{region '#Template'}
	{attribute 'Version' := '1.0.0.0'}
	{attribute 'Tags' := '"LCID": "1031", "Text": "H, General, HtgCir, Operating mode"'}
	{attribute 'Tags' := '"LCID": "1033", "Text": "H, General, HtgCir, Operating mode"'}
	{attribute 'Description' := '"LCID": "1031", "Text": "Betriebsart"'}
	{attribute 'Description' := '"LCID": "1033", "Text": "Operating mode"'}
{endregion}
FUNCTION_BLOCK FB_BA_H_OpMod EXTENDS FB_BA_View
VAR_INPUT
	bDst					: BOOL;
	bHtgLmt					: BOOL;
	bTWthLowLimit			: BOOL;
END_VAR
VAR_OUTPUT
	eOpMod					: E_BA_EnergyLvl;
	bRls					: BOOL;
END_VAR
VAR_INPUT CONSTANT
	OpModMan				: FB_BA_MV_Op;
	Sched					: FB_BA_SchedM;
	OpModPr					: FB_BA_MV_Op;								 
	Rls						: FB_BA_BV_Op;
END_VAR
VAR
	OpModSwi				: FB_BA_PrioSwi_UDI08;
	RlsMMux					: FB_BA_MMUX_B04;
END_VAR

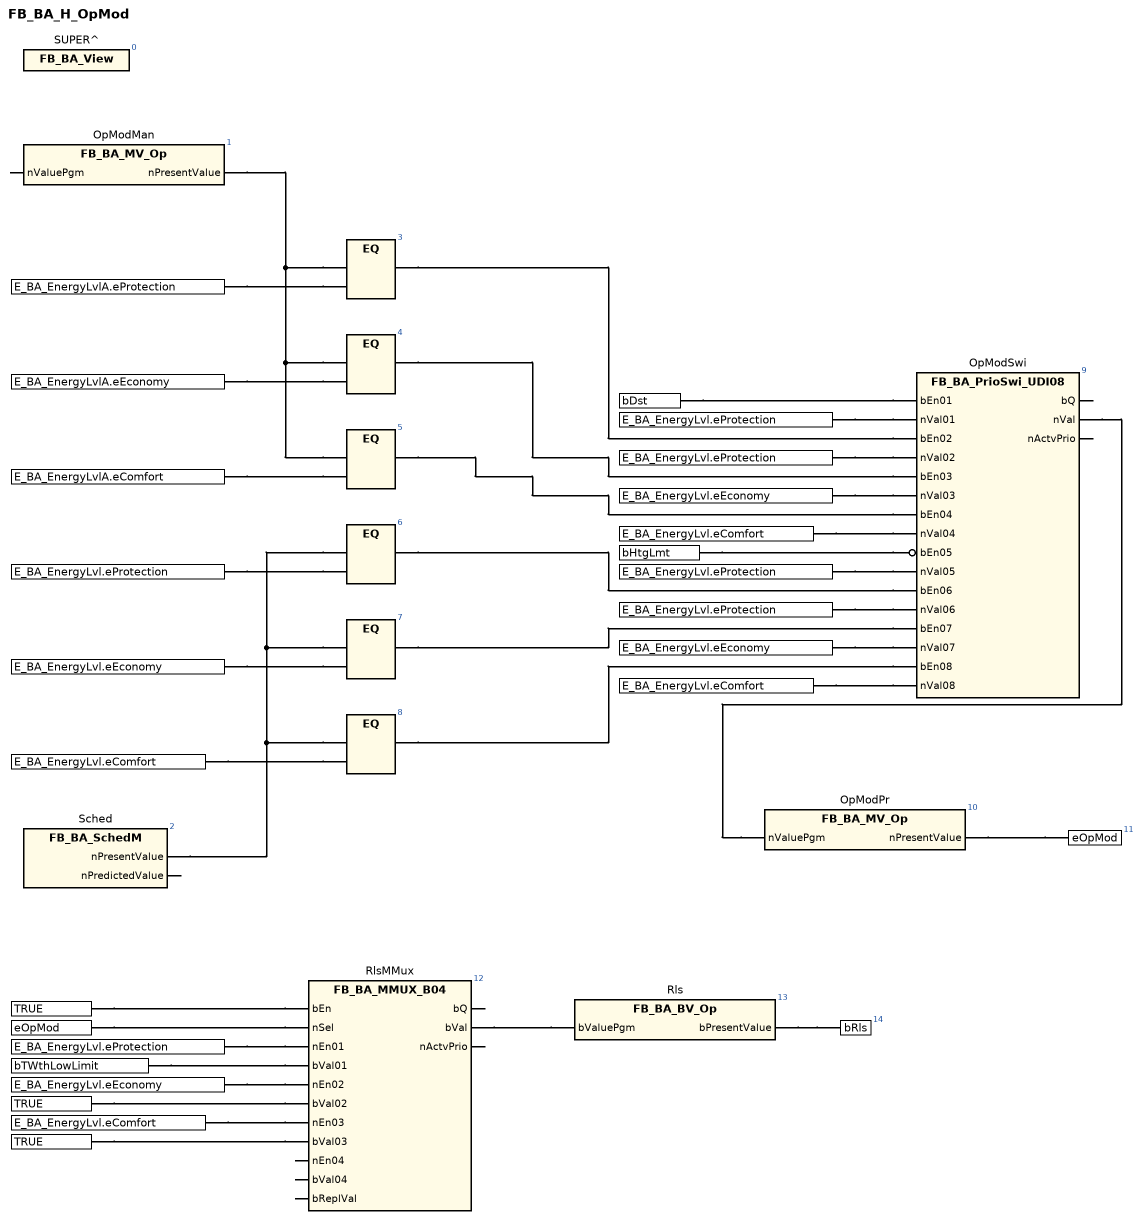
SUPER^(); // FB_BA_View
OpModMan(); // FB_BA_MV_Op
Sched(); // FB_BA_SchedM
OpModSwi(
    bEn01 := bDst,
    nVal01 := E_BA_EnergyLvl.eProtection,
    bEn02 := OpModMan.nPresentValue = E_BA_EnergyLvlA.eProtection,
    nVal02 := E_BA_EnergyLvl.eProtection,
    bEn03 := OpModMan.nPresentValue = E_BA_EnergyLvlA.eEconomy,
    nVal03 := E_BA_EnergyLvl.eEconomy,
    bEn04 := OpModMan.nPresentValue = E_BA_EnergyLvlA.eComfort,
    nVal04 := E_BA_EnergyLvl.eComfort,
    bEn05 := NOT bHtgLmt,
    nVal05 := E_BA_EnergyLvl.eProtection,
    bEn06 := Sched.nPresentValue = E_BA_EnergyLvl.eProtection,
    nVal06 := E_BA_EnergyLvl.eProtection,
    bEn07 := Sched.nPresentValue = E_BA_EnergyLvl.eEconomy,
    nVal07 := E_BA_EnergyLvl.eEconomy,
    bEn08 := Sched.nPresentValue = E_BA_EnergyLvl.eComfort,
    nVal08 := E_BA_EnergyLvl.eComfort); // FB_BA_PrioSwi_UDI08
OpModPr(nValuePgm := OpModSwi.nVal); // FB_BA_MV_Op
eOpMod := OpModPr.nPresentValue;
RlsMMux(
    bEn := TRUE,
    nSel := eOpMod,
    nEn01 := E_BA_EnergyLvl.eProtection,
    bVal01 := bTWthLowLimit,
    nEn02 := E_BA_EnergyLvl.eEconomy,
    bVal02 := TRUE,
    nEn03 := E_BA_EnergyLvl.eComfort,
    bVal03 := TRUE); // FB_BA_MMUX_B04
Rls(bValuePgm := RlsMMux.bVal); // FB_BA_BV_Op
bRls := Rls.bPresentValue;

METHOD FB_init : BOOL
VAR_INPUT
	bInitRetains : BOOL; // if TRUE, the retain variables are initialized (warm start / cold start)
	bInCopyCode : BOOL;  // if TRUE, the instance afterwards gets moved into the copy code (online change)
END_VAR
OpModMan.iParent		:= THIS^;
OpModMan.iLabel			:= LblCmpHeating.H_OpMod_OpModMan;							
OpModMan.sObjectName	:= '{Idx=01}';								 	 
OpModMan.aStateText[1]	:= txtEvent_Auto;
OpModMan.aStateText[2]	:= txtEvent_Protection;
OpModMan.aStateText[3]	:= txtEvent_Economy;
OpModMan.aStateText[4]	:= txtEvent_Comfort;
OpModMan.nValueRm		:= 1;

OpModPr.iParent			:= THIS^;
OpModPr.iLabel			:= LblCmpHeating.H_OpMod_OpModPr;							
OpModPr.sObjectName		:= '{Idx=01}';								 	 
OpModPr.aStateText[1]	:= txtEvent_Protection; 
OpModPr.aStateText[2]	:= txtEvent_Economy; 
OpModPr.aStateText[3]	:= txtEvent_Comfort; 
OpModPr.nValueRm		:= 1;

Rls.iParent				:= THIS^;
Rls.iLabel				:= LblCmpHeating.H_OpMod_Rls;	
Rls.sObjectName			:= '{Idx=01}';								 	 
Rls.sInactiveText		:= txtEvent_Off;
Rls.sActiveText			:= txtEvent_On;	
Rls.bValueRm			:= FALSE;								
Rls.eToggleMode 		:= E_BA_ToggleMode.eSwitch;	

Sched.iParent											:= THIS^;
Sched.iLabel											:= LblCmpHeating.H_OpMod_Sched;							
Sched.sObjectName										:= '{Idx=01}';								 	 
Sched.aStateText[1]										:= txtEvent_Protection;
Sched.aStateText[2]										:= txtEvent_Economy;
Sched.aStateText[3]										:= txtEvent_Comfort;
Sched.nPredictTime										:= 0;
Sched.nDefaultValue										:= E_BA_EnergyLvl.eProtection;
Sched.bWriteWeekly										:= FALSE;
//	Monday
Sched.aWeek[E_BA_Weekday.eMonday,1].eState				:= E_BA_SchedEntryState.eValue;
Sched.aWeek[E_BA_Weekday.eMonday,1].uValue.udiVal		:= E_BA_EnergyLvl.eComfort;
Sched.aWeek[E_BA_Weekday.eMonday,1].stTime.nHour		:= 6;
Sched.aWeek[E_BA_Weekday.eMonday,1].stTime.nMinute		:= 0;
Sched.aWeek[E_BA_Weekday.eMonday,1].stTime.nSecond		:= 0;
Sched.aWeek[E_BA_Weekday.eMonday,2].eState				:= E_BA_SchedEntryState.eValue;
Sched.aWeek[E_BA_Weekday.eMonday,2].uValue.udiVal		:= E_BA_EnergyLvl.eEconomy;
Sched.aWeek[E_BA_Weekday.eMonday,2].stTime.nHour		:= 20;
Sched.aWeek[E_BA_Weekday.eMonday,2].stTime.nMinute		:= 0;
Sched.aWeek[E_BA_Weekday.eMonday,2].stTime.nSecond		:= 0;
Sched.aWeek[E_BA_Weekday.eMonday,3].eState				:= E_BA_SchedEntryState.eValue;
Sched.aWeek[E_BA_Weekday.eMonday,3].uValue.udiVal		:= E_BA_EnergyLvl.eProtection;
Sched.aWeek[E_BA_Weekday.eMonday,3].stTime.nHour		:= 0;
Sched.aWeek[E_BA_Weekday.eMonday,3].stTime.nMinute		:= 0;
Sched.aWeek[E_BA_Weekday.eMonday,3].stTime.nSecond		:= 0;
//	Tuesday
Sched.aWeek[E_BA_Weekday.eTuesday,1].eState				:= E_BA_SchedEntryState.eValue;
Sched.aWeek[E_BA_Weekday.eTuesday,1].uValue.udiVal		:= E_BA_EnergyLvl.eComfort;
Sched.aWeek[E_BA_Weekday.eTuesday,1].stTime.nHour		:= 6;
Sched.aWeek[E_BA_Weekday.eTuesday,1].stTime.nMinute		:= 0;
Sched.aWeek[E_BA_Weekday.eTuesday,1].stTime.nSecond		:= 0;
Sched.aWeek[E_BA_Weekday.eTuesday,2].eState				:= E_BA_SchedEntryState.eValue;
Sched.aWeek[E_BA_Weekday.eTuesday,2].uValue.udiVal		:= E_BA_EnergyLvl.eEconomy;
Sched.aWeek[E_BA_Weekday.eTuesday,2].stTime.nHour		:= 20;
Sched.aWeek[E_BA_Weekday.eTuesday,2].stTime.nMinute		:= 0;
Sched.aWeek[E_BA_Weekday.eTuesday,2].stTime.nSecond		:= 0;
Sched.aWeek[E_BA_Weekday.eTuesday,3].eState				:= E_BA_SchedEntryState.eValue;
Sched.aWeek[E_BA_Weekday.eTuesday,3].uValue.udiVal		:= E_BA_EnergyLvl.eProtection;
Sched.aWeek[E_BA_Weekday.eTuesday,3].stTime.nHour		:= 0;
Sched.aWeek[E_BA_Weekday.eTuesday,3].stTime.nMinute		:= 0;
Sched.aWeek[E_BA_Weekday.eTuesday,3].stTime.nSecond		:= 0;
//	Wednesday
Sched.aWeek[E_BA_Weekday.eWednesday,1].eState			:= E_BA_SchedEntryState.eValue;
Sched.aWeek[E_BA_Weekday.eWednesday,1].uValue.udiVal	:= E_BA_EnergyLvl.eComfort;
Sched.aWeek[E_BA_Weekday.eWednesday,1].stTime.nHour		:= 6;
Sched.aWeek[E_BA_Weekday.eWednesday,1].stTime.nMinute	:= 0;
Sched.aWeek[E_BA_Weekday.eWednesday,1].stTime.nSecond	:= 0;
Sched.aWeek[E_BA_Weekday.eWednesday,2].eState			:= E_BA_SchedEntryState.eValue;
Sched.aWeek[E_BA_Weekday.eWednesday,2].uValue.udiVal	:= E_BA_EnergyLvl.eEconomy;
Sched.aWeek[E_BA_Weekday.eWednesday,2].stTime.nHour		:= 20;
Sched.aWeek[E_BA_Weekday.eWednesday,2].stTime.nMinute	:= 0;
Sched.aWeek[E_BA_Weekday.eWednesday,2].stTime.nSecond	:= 0;
Sched.aWeek[E_BA_Weekday.eWednesday,3].eState			:= E_BA_SchedEntryState.eValue;
Sched.aWeek[E_BA_Weekday.eWednesday,3].uValue.udiVal	:= E_BA_EnergyLvl.eProtection;
Sched.aWeek[E_BA_Weekday.eWednesday,3].stTime.nHour		:= 0;
Sched.aWeek[E_BA_Weekday.eWednesday,3].stTime.nMinute	:= 0;
Sched.aWeek[E_BA_Weekday.eWednesday,3].stTime.nSecond	:= 0;
//	Thursday
Sched.aWeek[E_BA_Weekday.eThursday,1].eState			:= E_BA_SchedEntryState.eValue;
Sched.aWeek[E_BA_Weekday.eThursday,1].uValue.udiVal		:=E_BA_EnergyLvl.eComfort;
Sched.aWeek[E_BA_Weekday.eThursday,1].stTime.nHour		:= 6;
Sched.aWeek[E_BA_Weekday.eThursday,1].stTime.nMinute	:= 0;
Sched.aWeek[E_BA_Weekday.eThursday,1].stTime.nSecond	:= 0;
Sched.aWeek[E_BA_Weekday.eThursday,2].eState			:= E_BA_SchedEntryState.eValue;
Sched.aWeek[E_BA_Weekday.eThursday,2].uValue.udiVal		:= E_BA_EnergyLvl.eEconomy;
Sched.aWeek[E_BA_Weekday.eThursday,2].stTime.nHour		:= 20;
Sched.aWeek[E_BA_Weekday.eThursday,2].stTime.nMinute	:= 0;
Sched.aWeek[E_BA_Weekday.eThursday,2].stTime.nSecond	:= 0;
Sched.aWeek[E_BA_Weekday.eThursday,3].eState			:= E_BA_SchedEntryState.eValue;
Sched.aWeek[E_BA_Weekday.eThursday,3].uValue.udiVal		:= E_BA_EnergyLvl.eProtection;
Sched.aWeek[E_BA_Weekday.eThursday,3].stTime.nHour		:= 0;
Sched.aWeek[E_BA_Weekday.eThursday,3].stTime.nMinute	:= 0;
Sched.aWeek[E_BA_Weekday.eThursday,3].stTime.nSecond	:= 0;
//	Friday
Sched.aWeek[E_BA_Weekday.eFriday,1].eState				:= E_BA_SchedEntryState.eValue;
Sched.aWeek[E_BA_Weekday.eFriday,1].uValue.udiVal		:= E_BA_EnergyLvl.eComfort;
Sched.aWeek[E_BA_Weekday.eFriday,1].stTime.nHour		:= 6;
Sched.aWeek[E_BA_Weekday.eFriday,1].stTime.nMinute		:= 0;
Sched.aWeek[E_BA_Weekday.eFriday,1].stTime.nSecond		:= 0;
Sched.aWeek[E_BA_Weekday.eFriday,2].eState				:= E_BA_SchedEntryState.eValue;
Sched.aWeek[E_BA_Weekday.eFriday,2].uValue.udiVal		:= E_BA_EnergyLvl.eEconomy;
Sched.aWeek[E_BA_Weekday.eFriday,2].stTime.nHour		:= 20;
Sched.aWeek[E_BA_Weekday.eFriday,2].stTime.nMinute		:= 0;
Sched.aWeek[E_BA_Weekday.eFriday,2].stTime.nSecond		:= 0;
Sched.aWeek[E_BA_Weekday.eFriday,3].eState				:= E_BA_SchedEntryState.eValue;
Sched.aWeek[E_BA_Weekday.eFriday,3].uValue.udiVal		:= E_BA_EnergyLvl.eProtection;
Sched.aWeek[E_BA_Weekday.eFriday,3].stTime.nHour		:= 0;
Sched.aWeek[E_BA_Weekday.eFriday,3].stTime.nMinute		:= 0;
Sched.aWeek[E_BA_Weekday.eFriday,3].stTime.nSecond		:= 0;
END_METHOD

END_FUNCTION_BLOCK

(* stored: Version 1.1.0.1, ProductVersion 3.1.4024.9
   POU FB_BA_H_OpMod: Id {21dadeb2-1455-42ac-9ff4-692d5cab4213}, SpecialFunc None
   Method FB_init: Id {75191e98-43ef-46b7-9ef5-6f27fa1df444} *)
